// Generates a boolean square wave with the given period
FUNCTION_BLOCK FB_SquareWave
VAR_INPUT
	tPeriod			: TIME;			// Period of the square wave
END_VAR
VAR_OUTPUT
	bSquareWave		: BOOL;			// Output square wave
END_VAR
VAR
	fbTimerOn		: TON;			// Timer FB
END_VAR

// Run FB
fbTimerOn();

IF fbTimerOn.Q THEN
	// Timer elapsed
	// Reset timer
	fbTimerOn.IN := FALSE;
	
	// Toggle output
	bSquareWave := NOT bSquareWave;
ELSE
	// Timer running
	// Set period
	fbTimerOn.PT := tPeriod / 2;
	
	// Enable timer
	fbTimerOn.IN := TRUE;	
END_IF

END_FUNCTION_BLOCK

(* stored: Version 1.1.0.1, ProductVersion 3.1.4024.12
   POU FB_SquareWave: Id {a4a642af-02d5-4cd3-bf05-19ed23282f75}, SpecialFunc None *)
